Staubli VAL3: start.pgx

program start()
  local num l_n
begin
  //Header begin
  //Description of Program
  // ATI Force Sensor
  // run as test of sensor
  // or use applicaiton as library
  //
  //Input parameters
  // none
  //
  //Output parameters
  // none
  //
  //Examples
  // run
  //
  //History
  // Creation: 10-Jul-2009, J Cook
  // Modification: 28-Feb-2013, yeyonglong
  //  description continued
  //
  //Header end
  call initialize("io:sAtiFs",l_n)
  taskCreateSync "readForce",0.004,bOverRun,loopReadForce()
  taskCreate "user",100,user()
end
